INTERFACE I_InputPort EXTENDS I_Disposable, I_EventEmitter, I_EventHandler, I_Serializable, I_HostMetadata

METHOD PUBLIC Accept
VAR_INPUT
	Visitor : I_InputPortVisitor;
END_VAR
END_METHOD

PROPERTY PUBLIC Connected : BOOL
GET
END_GET
END_PROPERTY

PROPERTY PUBLIC Data : I_Datatype
GET
END_GET
END_PROPERTY

METHOD PUBLIC Disconnect
END_METHOD

PROPERTY PUBLIC Name : T_MAXSTRING
GET
END_GET
END_PROPERTY

METHOD PUBLIC TryConnectTo : BOOL
VAR_INPUT
	OutputPort : I_OutputPort;
END_VAR
END_METHOD

END_INTERFACE

(* stored: Version 1.1.0.1, ProductVersion 3.1.4024.12
   Itf I_InputPort: Id {a332d5d8-4313-0a81-3b21-7ca5bb24d9de}
   Method Accept: Id {9c9c4d76-444e-06c3-0266-473605cb0e98}
   Property Connected: Id {d86180a6-ddfd-026f-3db3-6e01511f3c50}
   Get Get: Id {6f35463d-bc97-002d-31c1-16f2826c948b}
   Property Data: Id {b55d5762-c176-4884-bb3a-7b30355000fa}
   Get Get: Id {0ed95262-bbc6-48c8-a744-40d990b519bd}
   Method Disconnect: Id {94185341-941f-0d4c-1980-d9502ff11efe}
   Property Name: Id {d0512564-d953-055f-3d48-7ca34ce5cb91}
   Get Get: Id {f0059ff1-df44-0611-02fe-7795e4ae74ff}
   Method TryConnectTo: Id {1fbb9957-a7a2-0727-1cc1-31c666418ee0} *)
